//{attribute 'qualified_only'}
//{attribute 'strict'}
TYPE E_Station :
(
	eStation_none := 0,
	eStation_ST010_OvenA := 1,
	eStation_ST020_OvenB := 2,
	eStation_ST030_Handling := 3,
	eStation_ST040_Storage := 4,
	eStation_ST050_Mould := 5,
	
	/// has to be set to last index for array bounds!
	eStation_nMaxIdx
);
END_TYPE

(* stored: Version 1.1.0.1
   DUT E_Station: Id {05dfd324-689d-47f2-be0a-e8850ccd6d47} *)
